          Loop While (checkContinuously=false) expression=barreno_actual≤barrenos_menos1
            Folder Perforacion
              MoveL speed 100 mm/s, acceleration 500 mm/s^2 (useActiveTCP=true) feature=Base
                internos := interpolate_pose(Linea4_A, Linea4_B, barreno_actual/barrenos_menos1)
                Waypoint Waypoint (Variable): variable=internos
                'desbaste_inicial'
                bajada_broca := p[0,0,-0.024,0,0,0]
                bajada := p[0,0,0.024,0,0,0]
                MoveDirectionNode (selectedDirection=ZMinus toolParams=0.02, 0.015)
                  Until DISTANCE (allowActions=false deceleration=3 distanceNodeType=STOP) Distance=0.055; motionParameters(blendRadius=0)
                Popup Message (haltProgram=false message=punto contacto alanzdo inputType=Text)
                MoveDirectionNode (selectedDirection=ZPlus toolParams=0.003, 0.005)
                  Until DISTANCE (allowActions=false deceleration=3 distanceNodeType=STOP) Distance=0.001; motionParameters(blendRadius=0)
                Wait Sleep waitTime=0.3
                Set DigitalOutput pin=config_out[1]; digitalValue=1
                Wait Sleep waitTime=0.3
                Loop Counting (count=1) loopVariable(name=Loop_49)
                  bajar := pose_add(get_actual_tcp_pose(), bajada_broca)
                  Waypoint Waypoint (Variable): motionParameters(jointSpeed=1.047198 jointAcceleration=1.396263 cartesianSpeed=0.001 cartesianAcceleration=0.005); variable=bajar
                  subir := pose_sub(get_actual_tcp_pose(), bajada_broca)
                  Waypoint Waypoint (Variable): motionParameters(jointSpeed=1.047198 jointAcceleration=1.396263 cartesianSpeed=0.01 cartesianAcceleration=0.01); variable=subir
                  bajada_broca := pose_sub(bajada_broca, bajada)
                MoveDirectionNode (selectedDirection=ZPlus toolParams=0.03, 0.035)
                  Until DISTANCE (allowActions=false deceleration=3 distanceNodeType=STOP) Distance=0.06; motionParameters(blendRadius=0)
                Set DigitalOutput pin=config_out[1]; digitalValue=0
                barreno_actual := barreno_actual+1
                SuppressedNode
                  Call Quitar_broca
                SuppressedNode
                  Call Poner_broca
        Folder CD
          'desbaste_inicial'
          bajada_broca := p[0,0,-0.024,0,0,0]
          barrenos_menos1 := 8
          barreno_actual := 0
          Loop While (checkContinuously=false) expression=barreno_actual≤barrenos_menos1
            Folder Perforacion
              MoveL speed 100 mm/s, acceleration 500 mm/s^2 (useActiveTCP=true) feature=Base
                internos := interpolate_pose(Linea4_C, Linea4_D, barreno_actual/barrenos_menos1)
                Waypoint Waypoint (Variable): variable=internos
                'desbaste_inicial'
                bajada_broca := p[0,0,-0.024,0,0,0]
                bajada := p[0,0,0.024,0,0,0]
                MoveDirectionNode (selectedDirection=ZMinus toolParams=0.02, 0.015)
                  Until DISTANCE (allowActions=false deceleration=3 distanceNodeType=STOP) Distance=0.055; motionParameters(blendRadius=0)
                Popup Message (haltProgram=false message=punto contacto alanzdo inputType=Text)
                MoveDirectionNode (selectedDirection=ZPlus toolParams=0.003, 0.005)
                  Until DISTANCE (allowActions=false deceleration=3 distanceNodeType=STOP) Distance=0.001; motionParameters(blendRadius=0)
                Wait Sleep waitTime=0.3
                Set DigitalOutput pin=config_out[1]; digitalValue=1
                Wait Sleep waitTime=0.3
                Loop Counting (count=1) loopVariable(name=Loop_52)
                  bajar := pose_add(get_actual_tcp_pose(), bajada_broca)
                  Waypoint Waypoint (Variable): motionParameters(jointSpeed=1.047198 jointAcceleration=1.396263 cartesianSpeed=0.001 cartesianAcceleration=0.005); variable=bajar
                  subir := pose_sub(get_actual_tcp_pose(), bajada_broca)
                  Waypoint Waypoint (Variable): motionParameters(jointSpeed=1.047198 jointAcceleration=1.396263 cartesianSpeed=0.01 cartesianAcceleration=0.01); variable=subir
                  bajada_broca := pose_sub(bajada_broca, bajada)
                MoveDirectionNode (selectedDirection=ZPlus toolParams=0.03, 0.035)
                  Until DISTANCE (allowActions=false deceleration=3 distanceNodeType=STOP) Distance=0.06; motionParameters(blendRadius=0)
                Set DigitalOutput pin=config_out[1]; digitalValue=0
                barreno_actual := barreno_actual+1
                SuppressedNode
                  Call Quitar_broca
                SuppressedNode
                  Call Poner_broca
        Folder EF
          'desbaste_inicial'
          bajada_broca := p[0,0,-0.024,0,0,0]
          barrenos_menos1 := 8
          barreno_actual := 0
          Loop While (checkContinuously=false) expression=barreno_actual≤barrenos_menos1
            Folder Perforacion
              MoveL speed 100 mm/s, acceleration 500 mm/s^2 (useActiveTCP=true) feature=Base
                internos := interpolate_pose(Linea4_E, Linea4_F, barreno_actual/barrenos_menos1)
                Waypoint Waypoint (Variable): variable=internos
                'desbaste_inicial'
                bajada_broca := p[0,0,-0.024,0,0,0]
                bajada := p[0,0,0.024,0,0,0]
                MoveDirectionNode (selectedDirection=ZMinus toolParams=0.02, 0.015)
                  Until DISTANCE (allowActions=false deceleration=3 distanceNodeType=STOP) Distance=0.055; motionParameters(blendRadius=0)
                Popup Message (haltProgram=false message=punto contacto alanzdo inputType=Text)
                MoveDirectionNode (selectedDirection=ZPlus toolParams=0.003, 0.005)
                  Until DISTANCE (allowActions=false deceleration=3 distanceNodeType=STOP) Distance=0.001; motionParameters(blendRadius=0)
                Wait Sleep waitTime=0.3
                Set DigitalOutput pin=config_out[1]; digitalValue=1
                Wait Sleep waitTime=0.3
                Loop Counting (count=1) loopVariable(name=Loop_54)
                  bajar := pose_add(get_actual_tcp_pose(), bajada_broca)
                  Waypoint Waypoint (Variable): motionParameters(jointSpeed=1.047198 jointAcceleration=1.396263 cartesianSpeed=0.001 cartesianAcceleration=0.005); variable=bajar
                  subir := pose_sub(get_actual_tcp_pose(), bajada_broca)
                  Waypoint Waypoint (Variable): motionParameters(jointSpeed=1.047198 jointAcceleration=1.396263 cartesianSpeed=0.01 cartesianAcceleration=0.01); variable=subir
                  bajada_broca := pose_sub(bajada_broca, bajada)
                MoveDirectionNode (selectedDirection=ZPlus toolParams=0.03, 0.035)
                  Until DISTANCE (allowActions=false deceleration=3 distanceNodeType=STOP) Distance=0.06; motionParameters(blendRadius=0)
                Set DigitalOutput pin=config_out[1]; digitalValue=0
                barreno_actual := barreno_actual+1
                If barreno_actual≥barrenos_menos1
                  cambiar_broca := True
                SuppressedNode
                  Call Quitar_broca
                SuppressedNode
                  Call Poner_broca
      Popup Message (haltProgram=false message=Linea4 con full Terminada! inputType=Text)
    Folder 720
      Folder Broca_1
        Folder Linea5
          Folder Marcar_puntos
            MoveL speed 100 mm/s, acceleration 500 mm/s^2 (useActiveTCP=true) feature=Base
              Waypoint Home3: TCP in base x=-850.182 y=0 z=211.32 mm, rx=-2.0297 ry=2.3968 rz=0.0066 rad; joints [-14.374, -75.698, 98.757, -22.649, -284.037, -0.192] deg
              Waypoint Linea5_A: TCP in base x=-663.778 y=-510.056 z=80.075 mm, rx=3.1116 ry=-0.3921 rz=0.0087 rad; joints [15.224, -65.782, 99.916, -33.468, -339.581, -0.139] deg; TCP offset x=0.411 y=-218.298 z=37.994 mm, rx=1.558 ry=-0.1255 rz=0.1212 rad
              Waypoint Linea5_B: TCP in base x=-1154.197 y=-507.911 z=80.256 mm, rx=-2.6466 ry=1.68 rz=0.0007 rad; joints [13.333, -29.304, 35.323, -5.09, -290.95, -0.372] deg
          Folder AB
            'desbaste_inicial'
            bajada_broca := p[0,0,-0.008,0,0,0]
            barrenos_menos1 := 19
            barreno_actual := 0
            Loop While (checkContinuously=false) expression=barreno_actual≤barrenos_menos1
              Folder Perforacion
                MoveL speed 100 mm/s, acceleration 500 mm/s^2 (useActiveTCP=true) feature=Base
                  internos := interpolate_pose(Linea5_A, Linea5_B, barreno_actual/barrenos_menos1)
                  Waypoint Waypoint (Variable): variable=internos
                  'desbaste_inicial'
                  bajada_broca := p[0,0,-0.008,0,0,0]
                  bajada := p[0,0,0.008,0,0,0]
                  MoveDirectionNode (selectedDirection=ZMinus toolParams=0.007, 0.005)
                    Until TOOL_CONTACT_DETECTION (allowActions=false retraction=0 decelerationAcceleration=0.001 decelerationAngularAcceleration=34.906585)
                  Popup Message (haltProgram=false message=punto contacto alanzdo inputType=Text)
                  SuppressedNode
                    MoveDirectionNode (selectedDirection=ZPlus toolParams=0.003, 0.005)
                      Until DISTANCE (allowActions=false deceleration=3 distanceNodeType=STOP) Distance=0.002; motionParameters(blendRadius=0)
                  SuppressedNode
                    Wait Sleep waitTime=0.3
                  SuppressedNode
                    Set DigitalOutput pin=config_out[1]; digitalValue=1
                  SuppressedNode
                    Wait Sleep waitTime=0.3
                  SuppressedNode
                    Loop Counting (count=3) loopVariable(name=Loop_55)
                      bajar := pose_add(get_actual_tcp_pose(), bajada_broca)
                      Waypoint Waypoint (Variable): motionParameters(jointSpeed=1.047198 jointAcceleration=1.396263 cartesianSpeed=0.001 cartesianAcceleration=0.005); variable=bajar
                      subir := pose_sub(get_actual_tcp_pose(), bajada_broca)
                      Waypoint Waypoint (Variable): motionParameters(jointSpeed=1.047198 jointAcceleration=1.396263 cartesianSpeed=0.01 cartesianAcceleration=0.01); variable=subir
                      bajada_broca := pose_sub(bajada_broca, bajada)
                  MoveDirectionNode (selectedDirection=ZPlus toolParams=0.03, 0.035)
                    Until DISTANCE (allowActions=false deceleration=3 distanceNodeType=STOP) Distance=0.15; motionParameters(blendRadius=0)
                  Set DigitalOutput pin=config_out[1]; digitalValue=0
                  barreno_actual := barreno_actual+1
                  SuppressedNode
                    Call Quitar_broca
                  SuppressedNode
                    Call Poner_broca
          SuppressedNode
            Folder CD
              'desbaste_inicial'
              bajada_broca := p[0,0,-0.008,0,0,0]
              barrenos_menos1 := 8
              barreno_actual := 0
              Loop While (checkContinuously=false) expression=barreno_actual≤barrenos_menos1
                Folder Perforacion
                  MoveL speed 100 mm/s, acceleration 500 mm/s^2 (useActiveTCP=true) feature=Base
                    internos := interpolate_pose(Linea3_C, Linea3_D, barreno_actual/barrenos_menos1)
                    Waypoint Waypoint (Variable): variable=internos
                    'desbaste_inicial'
                    bajada_broca := p[0,0,-0.008,0,0,0]
                    bajada := p[0,0,0.008,0,0,0]
                    MoveDirectionNode (selectedDirection=ZMinus toolParams=0.02, 0.015)
                      Until DISTANCE (allowActions=false deceleration=3 distanceNodeType=STOP) Distance=0.055; motionParameters(blendRadius=0)
                    Popup Message (haltProgram=false message=punto contacto alanzdo inputType=Text)
                    MoveDirectionNode (selectedDirection=ZPlus toolParams=0.003, 0.005)
                      Until DISTANCE (allowActions=false deceleration=3 distanceNodeType=STOP) Distance=0.002; motionParameters(blendRadius=0)
                    Wait Sleep waitTime=0.3
                    Set DigitalOutput pin=config_out[1]; digitalValue=1
                    Wait Sleep waitTime=0.3
                    Loop Counting (count=3) loopVariable(name=Loop_57)
                      bajar := pose_add(get_actual_tcp_pose(), bajada_broca)
                      Waypoint Waypoint (Variable): motionParameters(jointSpeed=1.047198 jointAcceleration=1.396263 cartesianSpeed=0.001 cartesianAcceleration=0.005); variable=bajar
                      subir := pose_sub(get_actual_tcp_pose(), bajada_broca)
                      Waypoint Waypoint (Variable): motionParameters(jointSpeed=1.047198 jointAcceleration=1.396263 cartesianSpeed=0.01 cartesianAcceleration=0.01); variable=subir
                      bajada_broca := pose_sub(bajada_broca, bajada)
                    MoveDirectionNode (selectedDirection=ZPlus toolParams=0.03, 0.035)
                      Until DISTANCE (allowActions=false deceleration=3 distanceNodeType=STOP) Distance=0.06; motionParameters(blendRadius=0)
                    Set DigitalOutput pin=config_out[1]; digitalValue=0
                    barreno_actual := barreno_actual+1
                    SuppressedNode
                      Call Quitar_broca
                    SuppressedNode
                      Call Poner_broca
          SuppressedNode
            Folder EF
              'desbaste_inicial'
              bajada_broca := p[0,0,-0.008,0,0,0]
              barrenos_menos1 := 8
              barreno_actual := 0
              Loop While (checkContinuously=false) expression=barreno_actual≤barrenos_menos1
                Folder Perforacion
                  MoveL speed 100 mm/s, acceleration 500 mm/s^2 (useActiveTCP=true) feature=Base
                    internos := interpolate_pose(Linea3_E, Linea3_F, barreno_actual/barrenos_menos1)
                    Waypoint Waypoint (Variable): variable=internos
                    'desbaste_inicial'
                    bajada_broca := p[0,0,-0.008,0,0,0]
                    bajada := p[0,0,0.008,0,0,0]
                    MoveDirectionNode (selectedDirection=ZMinus toolParams=0.02, 0.015)
                      Until DISTANCE (allowActions=false deceleration=3 distanceNodeType=STOP) Distance=0.055; motionParameters(blendRadius=0)
                    Popup Message (haltProgram=false message=punto contacto alanzdo inputType=Text)
                    MoveDirectionNode (selectedDirection=ZPlus toolParams=0.003, 0.005)
                      Until DISTANCE (allowActions=false deceleration=3 distanceNodeType=STOP) Distance=0.002; motionParameters(blendRadius=0)
                    Wait Sleep waitTime=0.3
                    Set DigitalOutput pin=config_out[1]; digitalValue=1
                    Wait Sleep waitTime=0.3
                    Loop Counting (count=3) loopVariable(name=Loop_59)
                      bajar := pose_add(get_actual_tcp_pose(), bajada_broca)
                      Waypoint Waypoint (Variable): motionParameters(jointSpeed=1.047198 jointAcceleration=1.396263 cartesianSpeed=0.001 cartesianAcceleration=0.005); variable=bajar
                      subir := pose_sub(get_actual_tcp_pose(), bajada_broca)
                      Waypoint Waypoint (Variable): motionParameters(jointSpeed=1.047198 jointAcceleration=1.396263 cartesianSpeed=0.01 cartesianAcceleration=0.01); variable=subir
                      bajada_broca := pose_sub(bajada_broca, bajada)
                    MoveDirectionNode (selectedDirection=ZPlus toolParams=0.03, 0.035)
                      Until DISTANCE (allowActions=false deceleration=3 distanceNodeType=STOP) Distance=0.06; motionParameters(blendRadius=0)
                    Set DigitalOutput pin=config_out[1]; digitalValue=0
                    barreno_actual := barreno_actual+1
                    SuppressedNode
                      Call Quitar_broca
                    SuppressedNode
                      Call Poner_broca
        Popup Message (haltProgram=false message=Linea5 con chica Terminada! inputType=Text)
        Folder Linea6
          Folder Marcar_puntos
            MoveL speed 100 mm/s, acceleration 500 mm/s^2 (useActiveTCP=true) feature=Base
              Waypoint Home3: TCP in base x=-850.182 y=0 z=211.32 mm, rx=-2.0297 ry=2.3968 rz=0.0066 rad; joints [-14.374, -75.698, 98.757, -22.649, -284.037, -0.192] deg; TCP offset x=0.411 y=-218.298 z=37.994 mm, rx=1.558 ry=-0.1255 rz=0.1212 rad
              Waypoint Linea4_A: TCP in base x=-483.35 y=19.133 z=80.413 mm, rx=-2.0297 ry=2.3968 rz=0.0066 rad; joints [-34.857, -105.949, 143.743, -37.281, -304.535, -0.37] deg
              Waypoint Linea4_B: TCP in base x=-685.405 y=19.216 z=80.605 mm, rx=-2.0297 ry=2.3968 rz=0.0066 rad; joints [-21.02, -83.488, 123.782, -39.869, -290.712, -0.217] deg
              Waypoint Linea4_C: TCP in base x=-711.768 y=19.56 z=80.904 mm, rx=-2.0297 ry=2.3968 rz=0.0066 rad; joints [-20.032, -81.151, 120.968, -39.396, -289.723, -0.208] deg
              Waypoint Linea4_D: TCP in base x=-914.58 y=19.801 z=80.703 mm, rx=-2.0297 ry=2.3968 rz=0.0066 rad; joints [-14.612, -64.317, 97.516, -32.795, -284.295, -0.166] deg
              Waypoint Linea4_E: TCP in base x=-939.799 y=20.701 z=80.126 mm, rx=-2.0297 ry=2.3968 rz=0.0066 rad; joints [-14.202, -62.236, 94.311, -31.673, -283.882, -0.163] deg
              Waypoint Linea4_F: TCP in base x=-1143.008 y=20.924 z=80.361 mm, rx=-2.0297 ry=2.3968 rz=0.0066 rad; joints [-11.271, -44.369, 63.742, -18.977, -280.923, -0.147] deg
          Folder AB
            'desbaste_inicial'
            bajada_broca := p[0,0,-0.008,0,0,0]
            barrenos_menos1 := 8
            barreno_actual := 0
            Loop While (checkContinuously=false) expression=barreno_actual≤barrenos_menos1
              Folder Perforacion
                MoveL speed 100 mm/s, acceleration 500 mm/s^2 (useActiveTCP=true) feature=Base
                  internos := interpolate_pose(Linea4_A, Linea4_B, barreno_actual/barrenos_menos1)
                  Waypoint Waypoint (Variable): variable=internos
                  'desbaste_inicial'
                  bajada_broca := p[0,0,-0.008,0,0,0]
                  bajada := p[0,0,0.008,0,0,0]
                  MoveDirectionNode (selectedDirection=ZMinus toolParams=0.02, 0.015)
                    Until DISTANCE (allowActions=false deceleration=3 distanceNodeType=STOP) Distance=0.055; motionParameters(blendRadius=0)
                  Popup Message (haltProgram=false message=punto contacto alanzdo inputType=Text)
                  MoveDirectionNode (selectedDirection=ZPlus toolParams=0.003, 0.005)
                    Until DISTANCE (allowActions=false deceleration=3 distanceNodeType=STOP) Distance=0.002; motionParameters(blendRadius=0)
                  Wait Sleep waitTime=0.3
                  Set DigitalOutput pin=config_out[1]; digitalValue=1
                  Wait Sleep waitTime=0.3
                  Loop Counting (count=3) loopVariable(name=Loop_61)
                    bajar := pose_add(get_actual_tcp_pose(), bajada_broca)
                    Waypoint Waypoint (Variable): motionParameters(jointSpeed=1.047198 jointAcceleration=1.396263 cartesianSpeed=0.001 cartesianAcceleration=0.005); variable=bajar
                    subir := pose_sub(get_actual_tcp_pose(), bajada_broca)
                    Waypoint Waypoint (Variable): motionParameters(jointSpeed=1.047198 jointAcceleration=1.396263 cartesianSpeed=0.01 cartesianAcceleration=0.01); variable=subir
                    bajada_broca := pose_sub(bajada_broca, bajada)
                  MoveDirectionNode (selectedDirection=ZPlus toolParams=0.03, 0.035)
                    Until DISTANCE (allowActions=false deceleration=3 distanceNodeType=STOP) Distance=0.06; motionParameters(blendRadius=0)
                  Set DigitalOutput pin=config_out[1]; digitalValue=0
                  barreno_actual := barreno_actual+1
                  SuppressedNode
                    Call Quitar_broca
                  SuppressedNode
                    Call Poner_broca
          Folder CD
            'desbaste_inicial'
            bajada_broca := p[0,0,-0.008,0,0,0]
            barrenos_menos1 := 8
            barreno_actual := 0
            Loop While (checkContinuously=false) expression=barreno_actual≤barrenos_menos1
              Folder Perforacion
                MoveL speed 100 mm/s, acceleration 500 mm/s^2 (useActiveTCP=true) feature=Base
                  internos := interpolate_pose(Linea4_C, Linea4_D, barreno_actual/barrenos_menos1)
                  Waypoint Waypoint (Variable): variable=internos
                  'desbaste_inicial'
                  bajada_broca := p[0,0,-0.008,0,0,0]
                  bajada := p[0,0,0.008,0,0,0]
                  MoveDirectionNode (selectedDirection=ZMinus toolParams=0.02, 0.015)
                    Until DISTANCE (allowActions=false deceleration=3 distanceNodeType=STOP) Distance=0.055; motionParameters(blendRadius=0)
                  Popup Message (haltProgram=false message=punto contacto alanzdo inputType=Text)
                  MoveDirectionNode (selectedDirection=ZPlus toolParams=0.003, 0.005)
                    Until DISTANCE (allowActions=false deceleration=3 distanceNodeType=STOP) Distance=0.002; motionParameters(blendRadius=0)
                  Wait Sleep waitTime=0.3
                  Set DigitalOutput pin=config_out[1]; digitalValue=1
                  Wait Sleep waitTime=0.3
                  Loop Counting (count=3) loopVariable(name=Loop_63)
                    bajar := pose_add(get_actual_tcp_pose(), bajada_broca)
                    Waypoint Waypoint (Variable): motionParameters(jointSpeed=1.047198 jointAcceleration=1.396263 cartesianSpeed=0.001 cartesianAcceleration=0.005); variable=bajar
                    subir := pose_sub(get_actual_tcp_pose(), bajada_broca)
                    Waypoint Waypoint (Variable): motionParameters(jointSpeed=1.047198 jointAcceleration=1.396263 cartesianSpeed=0.01 cartesianAcceleration=0.01); variable=subir
                    bajada_broca := pose_sub(bajada_broca, bajada)
                  MoveDirectionNode (selectedDirection=ZPlus toolParams=0.03, 0.035)
                    Until DISTANCE (allowActions=false deceleration=3 distanceNodeType=STOP) Distance=0.06; motionParameters(blendRadius=0)
                  Set DigitalOutput pin=config_out[1]; digitalValue=0
                  barreno_actual := barreno_actual+1
                  SuppressedNode
                    Call Quitar_broca
                  SuppressedNode
                    Call Poner_broca
          Folder EF
            'desbaste_inicial'
            bajada_broca := p[0,0,-0.008,0,0,0]
            barrenos_menos1 := 8
            barreno_actual := 0
            Loop While (checkContinuously=false) expression=barreno_actual≤barrenos_menos1
              Folder Perforacion
                MoveL speed 100 mm/s, acceleration 500 mm/s^2 (useActiveTCP=true) feature=Base
                  internos := interpolate_pose(Linea4_E, Linea4_F, barreno_actual/barrenos_menos1)
                  Waypoint Waypoint (Variable): variable=internos
                  'desbaste_inicial'
                  bajada_broca := p[0,0,-0.008,0,0,0]
                  bajada := p[0,0,0.008,0,0,0]
                  MoveDirectionNode (selectedDirection=ZMinus toolParams=0.02, 0.015)
                    Until DISTANCE (allowActions=false deceleration=3 distanceNodeType=STOP) Distance=0.055; motionParameters(blendRadius=0)
                  Popup Message (haltProgram=false message=punto contacto alanzdo inputType=Text)
                  MoveDirectionNode (selectedDirection=ZPlus toolParams=0.003, 0.005)
                    Until DISTANCE (allowActions=false deceleration=3 distanceNodeType=STOP) Distance=0.002; motionParameters(blendRadius=0)
                  Wait Sleep waitTime=0.3
                  Set DigitalOutput pin=config_out[1]; digitalValue=1
                  Wait Sleep waitTime=0.3
                  Loop Counting (count=3) loopVariable(name=Loop_65)
                    bajar := pose_add(get_actual_tcp_pose(), bajada_broca)
                    Waypoint Waypoint (Variable): motionParameters(jointSpeed=1.047198 jointAcceleration=1.396263 cartesianSpeed=0.001 cartesianAcceleration=0.005); variable=bajar
                    subir := pose_sub(get_actual_tcp_pose(), bajada_broca)
                    Waypoint Waypoint (Variable): motionParameters(jointSpeed=1.047198 jointAcceleration=1.396263 cartesianSpeed=0.01 cartesianAcceleration=0.01); variable=subir
                    bajada_broca := pose_sub(bajada_broca, bajada)
                  MoveDirectionNode (selectedDirection=ZPlus toolParams=0.03, 0.035)
                    Until DISTANCE (allowActions=false deceleration=3 distanceNodeType=STOP) Distance=0.06; motionParameters(blendRadius=0)
                  Set DigitalOutput pin=config_out[1]; digitalValue=0
                  barreno_actual := barreno_actual+1
                  If barreno_actual≥barrenos_menos1
                    cambiar_broca := True
                  SuppressedNode
                    Call Quitar_broca
                  SuppressedNode
                    Call Poner_broca
        Popup Message (haltProgram=false message=Linea6 con chica Terminada! inputType=Text)
  'Subprogramas:'
SubProgram -> Quitar_broca
SubProgram -> Poner_broca
SubProgram Poner_broca (keepSynchronizedWithDisk=false)
  Folder Poner_broca
    If cambiar_broca≟ True  or iniciando_prog≟ True
      'Codigo de poner broca'
      Set DigitalOutput pin=ini_cambro_m289; digitalValue=0
      MoveL speed 250 mm/s, acceleration 1200 mm/s^2 (useActiveTCP=true) feature=Base
        Waypoint Precambio_broca: TCP in base x=0.83 y=461.518 z=287.521 mm, rx=-0.2218 ry=-3.132 rz=0.0004 rad; joints [-125.124, -120.118, 128.54, -7.699, -306.118, -0.232] deg; TCP offset x=0.411 y=-218.298 z=37.994 mm, rx=1.558 ry=-0.1255 rz=0.1212 rad
        Popup Warning (haltProgram=false message=Cambia a las siguientes brocas inputType=Text)
        Waypoint Dejar_broca: motionParameters(jointSpeed=1.047198 jointAcceleration=1.396263 cartesianSpeed=0.09 cartesianAcceleration=0.1); TCP in base x=0.824 y=461.516 z=12.952 mm, rx=-0.2218 ry=-3.132 rz=0.0004 rad; joints [-125.105, -101.29, 149.944, -47.99, -306.183, -0.134] deg; TCP offset x=0.411 y=-218.298 z=37.994 mm, rx=1.558 ry=-0.1255 rz=0.1212 rad
      Set DigitalOutput pin=ini_cambro_m289; digitalValue=1
      Wait Sleep waitTime=4
      Set DigitalOutput pin=ini_cambro_m289; digitalValue=0
      Wait Sleep waitTime=0.5
      Wait DigitalInput pin=fciclocarr_m292; digitalValue=0
      Wait Sleep waitTime=0.5
      MoveL speed 250 mm/s, acceleration 1200 mm/s^2 (useActiveTCP=true) feature=Base
        Waypoint Precambio_broca: motionParameters(jointSpeed=1.047198 jointAcceleration=1.396263 cartesianSpeed=0.09 cartesianAcceleration=0.1); TCP in base x=0.83 y=461.518 z=287.521 mm, rx=-0.2218 ry=-3.132 rz=0.0004 rad; joints [-125.124, -120.118, 128.54, -7.699, -306.118, -0.232] deg; TCP offset x=0.411 y=-218.298 z=37.994 mm, rx=1.558 ry=-0.1255 rz=0.1212 rad
      barrenos_hechos := 0
      iniciando_prog := False
      cambiar_broca := False
    If barrenos_hechos≟14
      If cambiar_broca≟ False
        'Codigo de poner broca'
        Set DigitalOutput pin=ini_cambro_m289; digitalValue=0
        MoveL speed 250 mm/s, acceleration 1200 mm/s^2 (useActiveTCP=true) feature=Base
          Waypoint Precambio_broca: TCP in base x=0.83 y=461.518 z=287.521 mm, rx=-0.2218 ry=-3.132 rz=0.0004 rad; joints [-125.124, -120.118, 128.54, -7.699, -306.118, -0.232] deg
          Waypoint Dejar_broca: motionParameters(jointSpeed=1.047198 jointAcceleration=1.396263 cartesianSpeed=0.09 cartesianAcceleration=0.1); TCP in base x=0.824 y=461.516 z=12.952 mm, rx=-0.2218 ry=-3.132 rz=0.0004 rad; joints [-125.105, -101.29, 149.944, -47.99, -306.183, -0.134] deg; TCP offset x=0.411 y=-218.298 z=37.994 mm, rx=1.558 ry=-0.1255 rz=0.1212 rad
        Set DigitalOutput pin=ini_cambro_m289; digitalValue=1
        Wait Sleep waitTime=4
        Set DigitalOutput pin=ini_cambro_m289; digitalValue=0
        Wait Sleep waitTime=0.5
        Wait DigitalInput pin=fciclocarr_m292; digitalValue=0
        Wait Sleep waitTime=0.5
        MoveL speed 250 mm/s, acceleration 1200 mm/s^2 (useActiveTCP=true) feature=Base
          Waypoint Precambio_broca: motionParameters(jointSpeed=1.047198 jointAcceleration=1.396263 cartesianSpeed=0.09 cartesianAcceleration=0.1); TCP in base x=0.83 y=461.518 z=287.521 mm, rx=-0.2218 ry=-3.132 rz=0.0004 rad; joints [-125.124, -120.118, 128.54, -7.699, -306.118, -0.232] deg; TCP offset x=0.411 y=-218.298 z=37.994 mm, rx=1.558 ry=-0.1255 rz=0.1212 rad
        barrenos_hechos := 0
      Else 
        'Codigo de poner broca'
        Set DigitalOutput pin=ini_cambro_m289; digitalValue=0
        MoveL speed 250 mm/s, acceleration 1200 mm/s^2 (useActiveTCP=true) feature=Base
          Waypoint Precambio_broca: TCP in base x=0.83 y=461.518 z=287.521 mm, rx=-0.2218 ry=-3.132 rz=0.0004 rad; joints [-125.124, -120.118, 128.54, -7.699, -306.118, -0.232] deg
          Popup Warning (haltProgram=false message=Cambia a las siguientes brocas inputType=Text)
          Waypoint Dejar_broca: motionParameters(jointSpeed=1.047198 jointAcceleration=1.396263 cartesianSpeed=0.09 cartesianAcceleration=0.1); TCP in base x=0.824 y=461.516 z=12.952 mm, rx=-0.2218 ry=-3.132 rz=0.0004 rad; joints [-125.105, -101.29, 149.944, -47.99, -306.183, -0.134] deg; TCP offset x=0.411 y=-218.298 z=37.994 mm, rx=1.558 ry=-0.1255 rz=0.1212 rad
        Set DigitalOutput pin=ini_cambro_m289; digitalValue=1
        Wait Sleep waitTime=4
        Set DigitalOutput pin=ini_cambro_m289; digitalValue=0
        Wait Sleep waitTime=0.5
        Wait DigitalInput pin=fciclocarr_m292; digitalValue=0
        Wait Sleep waitTime=0.5
        MoveL speed 250 mm/s, acceleration 1200 mm/s^2 (useActiveTCP=true) feature=Base
          Waypoint Precambio_broca: motionParameters(jointSpeed=1.047198 jointAcceleration=1.396263 cartesianSpeed=0.09 cartesianAcceleration=0.1); TCP in base x=0.83 y=461.518 z=287.521 mm, rx=-0.2218 ry=-3.132 rz=0.0004 rad; joints [-125.124, -120.118, 128.54, -7.699, -306.118, -0.232] deg; TCP offset x=0.411 y=-218.298 z=37.994 mm, rx=1.558 ry=-0.1255 rz=0.1212 rad
        barrenos_hechos := 0
        iniciando_prog := False
        cambiar_broca := False
SubProgram Quitar_broca (keepSynchronizedWithDisk=false)
  Folder Quitar_broca
    barrenos_hechos := barrenos_hechos+1
    If barrenos_hechos≟14 or cambiar_broca≟ True
      'Codigo de quitar broca'
      MoveL speed 250 mm/s, acceleration 1200 mm/s^2 (useActiveTCP=true) feature=Base
        MoveDirectionNode (selectedDirection=ZPlus)
          Until DISTANCE (allowActions=false deceleration=3 distanceNodeType=STOP) Distance=0.3; motionParameters(blendRadius=0)
        If eje7≟3
          Waypoint Precambio_broca: TCP in base x=0.83 y=461.518 z=287.521 mm, rx=-0.2218 ry=-3.132 rz=0.0004 rad; joints [-125.124, -120.118, 128.54, -7.699, -306.118, -0.232] deg
        Waypoint Precambio_broca: TCP in base x=0.83 y=461.518 z=287.521 mm, rx=-0.2218 ry=-3.132 rz=0.0004 rad; joints [-125.124, -120.118, 128.54, -7.699, -306.118, -0.232] deg
        Waypoint Dejar_broca: motionParameters(jointSpeed=1.047198 jointAcceleration=1.396263 cartesianSpeed=0.09 cartesianAcceleration=0.1); TCP in base x=0.824 y=461.516 z=12.952 mm, rx=-0.2218 ry=-3.132 rz=0.0004 rad; joints [-125.105, -101.29, 149.944, -47.99, -306.183, -0.134] deg; TCP offset x=0.411 y=-218.298 z=37.994 mm, rx=1.558 ry=-0.1255 rz=0.1212 rad
      Set DigitalOutput pin=outputbroc_m291; digitalValue=1
      Wait Sleep waitTime=4
      Set DigitalOutput pin=outputbroc_m291; digitalValue=0
      Wait Sleep waitTime=0.5
      Wait DigitalInput pin=fciclocarr_m292; digitalValue=0
      Wait Sleep waitTime=0.5
      MoveL speed 250 mm/s, acceleration 1200 mm/s^2 (useActiveTCP=true) feature=Base
        Waypoint Precambio_broca: motionParameters(jointSpeed=1.047198 jointAcceleration=1.396263 cartesianSpeed=0.09 cartesianAcceleration=0.1); TCP in base x=0.83 y=461.518 z=287.521 mm, rx=-0.2218 ry=-3.132 rz=0.0004 rad; joints [-125.124, -120.118, 128.54, -7.699, -306.118, -0.232] deg; TCP offset x=0.411 y=-218.298 z=37.994 mm, rx=1.558 ry=-0.1255 rz=0.1212 rad
      Set DigitalOutput pin=avancarrusel_m7; digitalValue=1
      Wait Sleep waitTime=1
      Set DigitalOutput pin=avancarrusel_m7; digitalValue=0
      Wait Sleep waitTime=0.1
